FUNCTION_BLOCK F_TIME_IN_S_TO_LINT (* Convert TIME to LINT in seconds *)
  (* Standard: 61499-1; Description: Copyright (c) 2019 TU Wien/ACIN This program and the accompanying materials are made available under the terms of the Eclipse Public License 2.0 which is available at https://www.eclipse.org/legal/epl-2.0/ SPDX-License-Identifier: EPL-2.0 *)
  (* Version 1.0, 2019-07-08, Martin Melik Merkumians, TU Wien/ACIN *)
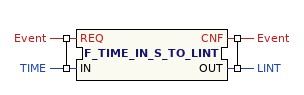
  EVENT_INPUT
    REQ WITH IN; (* Normal Execution Request *)
  END_EVENT
  EVENT_OUTPUT
    CNF WITH OUT; (* Execution Confirmation *)
  END_EVENT
  VAR_INPUT
    IN : TIME;
  END_VAR
  VAR_OUTPUT
    OUT : LINT;
  END_VAR
  ALGORITHM REQ IN ST:
OUT := TIME_IN_S_TO_LINT(IN);
  END_ALGORITHM
END_FUNCTION_BLOCK
